{attribute 'qualified_only'}
{attribute 'strict'}
{attribue 'to_string}
TYPE ePowerControlType :
(
	Current := 0,
	Power	:=1,
	Both	:= 2
);
END_TYPE

(* stored: Version 1.1.0.1, ProductVersion 3.1.4026.18
   DUT ePowerControlType: Id {ebc349c1-966c-4657-b258-4559a55d8ee2} *)
